# B&R Automation Studio project lab1v1
Automation Studio 4.5.2.102

## Configuration Config1

### Hardware
```
4PP065_0571_P74 : 4PP065.0571-P74 v1.1.2.0
  Connector IF5:
    ActivateDevice = 1
  ConfigurationID = lab1v1_Config1
  Simulation = 1
```

## Logical view

Binary libraries used (declarations not repeated): operator, runtime, astime, AsIecCon

### Library Logical/Libraries/Library (ANSIC)

#### Library.fun - Exported functions and function blocks
```iecst
{REDUND_ERROR} {REDUND_UNREPLICABLE} FUNCTION_BLOCK FB_Motor (*TODO: Add your comment here*) (*$GROUP=User,$CAT=User,$GROUPICON=User.png,$CATICON=User.png*)
	VAR_INPUT
		u : {REDUND_UNREPLICABLE} REAL;
	END_VAR
	VAR_OUTPUT
		w : {REDUND_UNREPLICABLE} REAL;
		phi : {REDUND_UNREPLICABLE} REAL;
	END_VAR
	VAR
		integrator : {REDUND_UNREPLICABLE} FB_Integrator;
		Tm : {REDUND_UNREPLICABLE} REAL;
		ke : {REDUND_UNREPLICABLE} REAL;
		dt : {REDUND_UNREPLICABLE} REAL;
	END_VAR
END_FUNCTION_BLOCK

{REDUND_ERROR} FUNCTION_BLOCK FB_Integrator (*TODO: Add your comment here*) (*$GROUP=User,$CAT=User,$GROUPICON=User.png,$CATICON=User.png*)
	VAR_INPUT
		in : {REDUND_UNREPLICABLE} REAL;
	END_VAR
	VAR
		out : {REDUND_UNREPLICABLE} REAL;
		dt : {REDUND_UNREPLICABLE} REAL;
		prev_value : REAL;
	END_VAR
END_FUNCTION_BLOCK

{REDUND_ERROR} FUNCTION_BLOCK FB_Regulator (*TODO: Add your comment here*) (*$GROUP=User,$CAT=User,$GROUPICON=User.png,$CATICON=User.png*)
	VAR_INPUT
		e : {REDUND_UNREPLICABLE} REAL;
	END_VAR
	VAR_OUTPUT
		u : REAL;
	END_VAR
	VAR
		integrator : FB_Integrator;
		k_p : REAL;
		k_i : REAL;
		iyOld : REAL;
		dt : REAL;
		max_abs_value : REAL;
	END_VAR
END_FUNCTION_BLOCK
```

#### FB_Integrator.c
```c
#include <bur/plctypes.h>
#ifdef __cplusplus
  extern "C"
  {
#endif
#include "Library.h"
#ifdef __cplusplus
  };
#endif

void FB_Integrator(struct FB_Integrator* inst)
{
	inst->out = inst->dt * inst->in + inst->prev_value;
	inst->prev_value = inst->out;
}
```

#### FB_Motor.c
```c
#include <bur/plctypes.h>
#ifdef __cplusplus
  extern "C"
  {
#endif
#include "Library.h"
#ifdef __cplusplus
  };
#endif

void FB_Motor(struct FB_Motor* inst)
{
	REAL a = inst->u / inst->ke - inst->w;
	REAL b = a / inst->Tm;

	inst->integrator.in = b;
	FB_Integrator(&inst->integrator);

	inst->w = inst->integrator.out;
}
```

#### FB_Regulator.c
```c
#include <bur/plctypes.h>
#ifdef __cplusplus
  extern "C"
  {
#endif
#include "Library.h"
#ifdef __cplusplus
  };
#endif

void FB_Regulator(struct FB_Regulator* inst)
{
	//vremennye peremennye
	REAL a = inst->e * inst ->k_p;
	REAL b = inst->e * inst ->k_i;
  	//ogranichenie napryazeniya

	a = a > inst->max_abs_value ? inst ->max_abs_value : a;
	a = a < -inst ->max_abs_value ? -inst ->max_abs_value : a;

	inst->integrator.in = b + inst->iyOld;

	FB_Integrator(&inst->integrator);

	REAL sum = a + inst->integrator.out;
	inst->u = sum;

	//ogranichenie napryazeniya
	inst->u = inst->u > inst->max_abs_value ? inst->max_abs_value : inst->u;
	inst->u = inst->u < -inst->max_abs_value ? inst->max_abs_value : inst->u;

	inst->iyOld = inst->u - sum;
}
```

### Program Logical/Program (ANSIC)

#### Variables.var - Local variables
```iecst
VAR
	Enable : BOOL;
	counter : INT;
	fb_motor1 : FB_Motor;
	fb_controller : FB_Regulator;
	fb_motor2 : FB_Motor;
	Speed : REAL;
END_VAR
```

Listed in the project but not available here: Logical/Libraries/Library/Types.typ, Logical/Libraries/Library/Constants.var, Logical/Program/Main.c, Logical/Program/Types.typ
